{region '#Template'}
	{attribute 'Version' := '5.0.0.0'}
	{attribute 'Tags' := '"LCID": "1031", "Text": "Universal, Motor, Aggregate"'}
	{attribute 'Tags' := '"LCID": "1033", "Text": "Universal, Motor, Aggregate"'}
	{attribute 'Using' := '"Type": "Template", "URI": "EC_ID"'}
	{attribute 'Using' := '"Type": "Template", "URI": "BA2_Param"'}
	{attribute 'Description' := '"LCID": "1031", "Text": "Motor modulierend mit Regler erweitert"'}
	{attribute 'Description' := '"LCID": "1033", "Text": "Motor modulating with controller extended"'}
{endregion}		 
FUNCTION_BLOCK FB_BA_MotCtlExt EXTENDS FB_BA_MotCtl
VAR_INPUT CONSTANT
	ThOvrld			: FB_BA_BI_Raw;							
	MntnSwi			: FB_BA_BI_Raw;
END_VAR
VAR
END_VAR

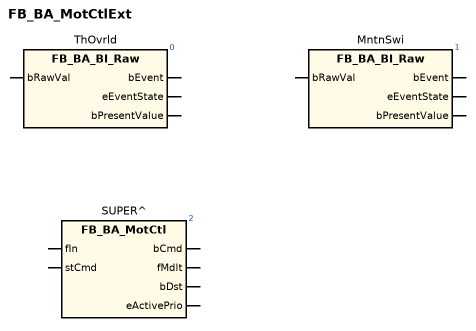
ThOvrld(); // FB_BA_BI_Raw
MntnSwi(); // FB_BA_BI_Raw
SUPER^(); // FB_BA_MotCtl

METHOD FB_init : BOOL
VAR_INPUT
	bInitRetains : BOOL; // if TRUE, the retain variables are initialized (warm start / cold start)
	bInCopyCode : BOOL;  // if TRUE, the instance afterwards gets moved into the copy code (online change)
END_VAR
ThOvrld.iParent						:= THIS^;
ThOvrld.iLabel						:= LblFun_Fault;  
ThOvrld.ePolarity					:= E_BA_Polarity.eReverse;
ThOvrld.sActiveText 				:= txtEvent_Triggered;
ThOvrld.sInactiveText 				:= txtEvent_Normal;
ThOvrld.nEventClassID				:= EC_ID.NC30;
ThOvrld.stTimeDelay.nToNormal		:= BA2_Param.nDefTimeDelay_ToNormal;
ThOvrld.stTimeDelay.nToAbnormal		:= BA2_Param.nDefTimeDelay_ToAbnormal;
ThOvrld.bAlarmValue					:= TRUE;
ThOvrld.aEventTransitionText[1]		:= txtEvent_Triggered;
ThOvrld.aEventTransitionText[2]		:= txtEvent_Error;
ThOvrld.aEventTransitionText[3]		:= txtEvent_Normal;
ThOvrld.bEventDetectionEnable		:= TRUE;
ThOvrld.eEnPlantLock				:= E_BA_LockPriority.eLocalMedium;	

MntnSwi.iParent						:= THIS^;
MntnSwi.iLabel						:= LblFun_MaintenanceMessage;  
MntnSwi.ePolarity					:= E_BA_Polarity.eReverse;
MntnSwi.sActiveText 				:= txtEvent_Maintenace;
MntnSwi.sInactiveText 				:= txtEvent_Normal;
MntnSwi.nEventClassID				:= EC_ID.NC50;
MntnSwi.stTimeDelay.nToNormal		:= BA2_Param.nDefTimeDelay_ToNormal;
MntnSwi.stTimeDelay.nToAbnormal		:= BA2_Param.nDefTimeDelay_ToAbnormal;
MntnSwi.bAlarmValue					:= TRUE;
MntnSwi.aEventTransitionText[1]		:= txtEvent_Disturb;
MntnSwi.aEventTransitionText[2]		:= txtEvent_None;
MntnSwi.aEventTransitionText[3]		:= txtEvent_Normal;
MntnSwi.bEventDetectionEnable		:= TRUE;
MntnSwi.eEnPlantLock				:= E_BA_LockPriority.eLocalMedium;
END_METHOD

END_FUNCTION_BLOCK

(* stored: Version 1.1.0.1, ProductVersion 3.1.4024.12
   POU FB_BA_MotCtlExt: Id {71303cc5-75db-442b-86eb-6495805e1989}, SpecialFunc None
   Method FB_init: Id {4a5ad6bc-ecfd-46a4-8c6d-838a8355bf7b} *)
